// TIA Portal V17 export
// export: Created 2023-02-13T11:16:51.9785059Z, ExportSetting WithDefaults, DisplayName Totally Integrated Automation Portal, DisplayVersion V17, DisplayName TIA Portal Openness, DisplayVersion V17, DisplayName TIA Portal Teamcenter Gateway, DisplayVersion V17, DisplayName TIA Portal Version Control Interface, DisplayVersion V17, DisplayName SINAMICS Startdrive Advanced, DisplayVersion V17, DisplayName SINAMICS Startdrive G130, G150, S120, S150, SINAMICS MV, S210, DisplayVersion V17, DisplayName SINAMICS Startdrive G110M, G120, G120C, G120D, G120P, G115D, DisplayVersion V17, DisplayName STEP 7 Professional, DisplayVersion V17, DisplayName STEP 7 Safety, DisplayVersion V17, DisplayName WinCC Professional, DisplayVersion V17
FUNCTION_BLOCK "BFT_Type5"   // FB355, LAD
{ S7_Optimized_Access := 'TRUE' }
VERSION : 0.1
// Buffer Tank Vinegar
// stored: AutoNumber false, IsIECCheckEnabled false, IsRetainMemResEnabled false, MemoryReserve 100, SetENOAutomatically false, UDAEnableTagReadback false
   VAR_INPUT
      "IN_FBAV.01" : Bool := FALSE;   // Tank Flushing Water Valve
      "IN_FBAV.02" : Bool := FALSE;   // Tank CIP Top Inlet Valve
      "IN_FBAV.03" : Bool := FALSE;   // Tank Tank Outlet Valve
      "IN_FBSV.01" : Bool := FALSE;   // SV Diaphragm Pump Inlet Material
      IN_LT01 : Real;   // Tank Level Transmitter
      "IN_FBP.01" : Bool := FALSE;   // Transfer Pump
      "IN_P.01-Speed" : Real;   // Transfer Pump AV Speed
      DosePumpSpeed : Real;
      "DoseON-OFF" : Bool := FALSE;
      "DosePumpON-OFF" : Bool := FALSE;
      CIPPulse : Bool := FALSE;
      CIP_Supply_ON : Bool;
      CIP_Busy : Bool;   // Line CIP in USE
      LineTrf_OK : Bool := FALSE;
      LineFlush_OK : Bool;
      LCS_Start : Bool;   // Start Command from LCS
      LCS_Stop : Bool;   // Stop Command from LCS
   END_VAR
   VAR_OUTPUT
      "OUT_AV.01" : Bool := FALSE;   // Tank Flushing Water Valve
      "OUT_AV.02" : Bool := FALSE;   // Tank CIP Top Inlet Valve
      "OUT_AV.03" : Bool := FALSE;   // Tank Tank Outlet Valve
      "OUT_AV.06" : Bool := FALSE;   // Tank Tank Outlet Valve
      "OUT_P.01" : Bool := FALSE;   // Transfer Pump
      "OUT_P.01-Speed" : Real;   // Transfer Pump AV Speed
      "OUT_SV.01" : Bool := FALSE;   // SV Diaphragm Pump Inlet Material
      OUT_CIPTank_AVOpen : Bool;
   END_VAR
   VAR
      Cmd { ExternalVisible := 'False'} : Struct
         Inload { ExternalVisible := 'False'} : Bool;   // Start Loading
         RaadyForMix { ExternalVisible := 'False'} : Bool;   // Tank Ready for Blending
         Tank_CIP_Req { ExternalVisible := 'False'} : Bool;
         Flush_Select { ExternalVisible := 'False'} : Byte;
         Flushing { ExternalVisible := 'False'} : Bool;   // Water Flushing
      END_STRUCT;
      Param { ExternalVisible := 'False'} : Struct
         SP_Level_LL { ExternalVisible := 'False'} : Real := 10.0;
         SP_Level_ML { ExternalVisible := 'False'} : Real := 80.0;
         SP_Level_HL { ExternalVisible := 'False'} : Real := 100.0;
         L_Hi_Lim { ExternalVisible := 'False'} : Real := 100.0;
         L_Lo_Lim { ExternalVisible := 'False'} : Real := 0.0;
         L_Hys { ExternalVisible := 'False'} : Real := 5.0;
         FlushingTime { ExternalVisible := 'False'} : Time := T#10s;
         CIP_Trf_SP_Speed { ExternalVisible := 'False'} : Real := 80.0;
         CIP_Ret_ON_SP { ExternalVisible := 'False'} : Real := 5.0;
         CIP_Ret_OFF_SP { ExternalVisible := 'False'} : Real;
      END_STRUCT;
      State { ExternalVisible := 'False'} : Struct   // Tank in loading state
         Tank_inloading { ExternalVisible := 'False'} : Bool;
         Tank_inRawDose { ExternalVisible := 'False'} : Bool;
         Tank_inCIP { ExternalVisible := 'False'} : Bool;
         Line_inCIP { ExternalVisible := 'False'} : Bool;
         Flushing { ExternalVisible := 'False'} : Bool;
         Tank_LL { ExternalVisible := 'False'} : Bool;
         Tank_ML { ExternalVisible := 'False'} : Bool;
         Tank_HL { ExternalVisible := 'False'} : Bool;
         Inload_Enable { ExternalVisible := 'False'} : Bool;
         Tank_CIP_Enable { ExternalVisible := 'False'} : Bool;
         Line_CIP_Enable { ExternalVisible := 'False'} : Bool;
         Flushing_Enable { ExternalVisible := 'False'} : Bool;
         Flush_selected { ExternalVisible := 'False'} : Byte;
         CIP_Request_OK { ExternalVisible := 'False'} : Bool;
         CIP_ReturnON { ExternalVisible := 'False'} : Bool;
         Ready_For_Transfer { ExternalVisible := 'False'} : Bool;   // Tank Ready for Transfer to Blending
         Ready_For_Transfer_EN { ExternalVisible := 'False'} : Bool;   // Tank Ready for Transfer to Blending
         Transfer_to_Blend { ExternalVisible := 'False'} : Bool;
         Status { ExternalVisible := 'False'} : Int;
      END_STRUCT;
      alwaysON : Bool;
      L_Hys_Abs : Real;
      Hys_Level_HL : Real;
      Hys_Level_ML : Real;
      Hys_Level_LL : Real;
      r : Struct
         PosE1 : Bool;
         PosE2 : Bool;
         PosE3 : Bool;
         PosE4 : Bool;
         PosE5 : Bool;
         PosE6 : Bool;
         PosE7 : Bool;
         PosE8 : Bool;
         PosE9 : Bool;
         PosE10 : Bool;
         PosE11 : Bool;
         PosE12 : Bool;
         PosE13 : Bool;
         PosE14 : Bool;
         PosE15 : Bool;
         PosE16 : Bool;
         PosE17 : Bool;
         PosE18 : Bool;
         PosE19 : Bool;
         PosE20 : Bool;
         PosE21 : Bool;
         PosE22 : Bool;
         PosE23 : Bool;
         PosE24 : Bool;
         PosE25 : Bool;
         PosE26 : Bool;
         PosE27 : Bool;
         PosE28 : Bool;
         PosE29 : Bool;
         PosE30 : Bool;
         PosE31 : Bool;
         PosE32 : Bool;
      END_STRUCT;
      Actuator : Struct
         AV_Outlet : Bool;
         TransferPump : Bool;
         FlushPump : Bool;
         CV_Steam : Bool;
         Pump : Bool;
         Agitator_level : Bool;
         LCS_OnOff : Bool;
      END_STRUCT;
      FlushingTim : TON_TIME;
   END_VAR
   VAR_TEMP   // added for the SCL form of the ladder/FBD networks
      _w1 : Bool;
      _w2 : Bool;
      _w3 : Bool;
      _w4 : Bool;
      _w5 : Bool;
      _w6 : Bool;
   END_VAR
BEGIN

REGION Network 1: Always_ON
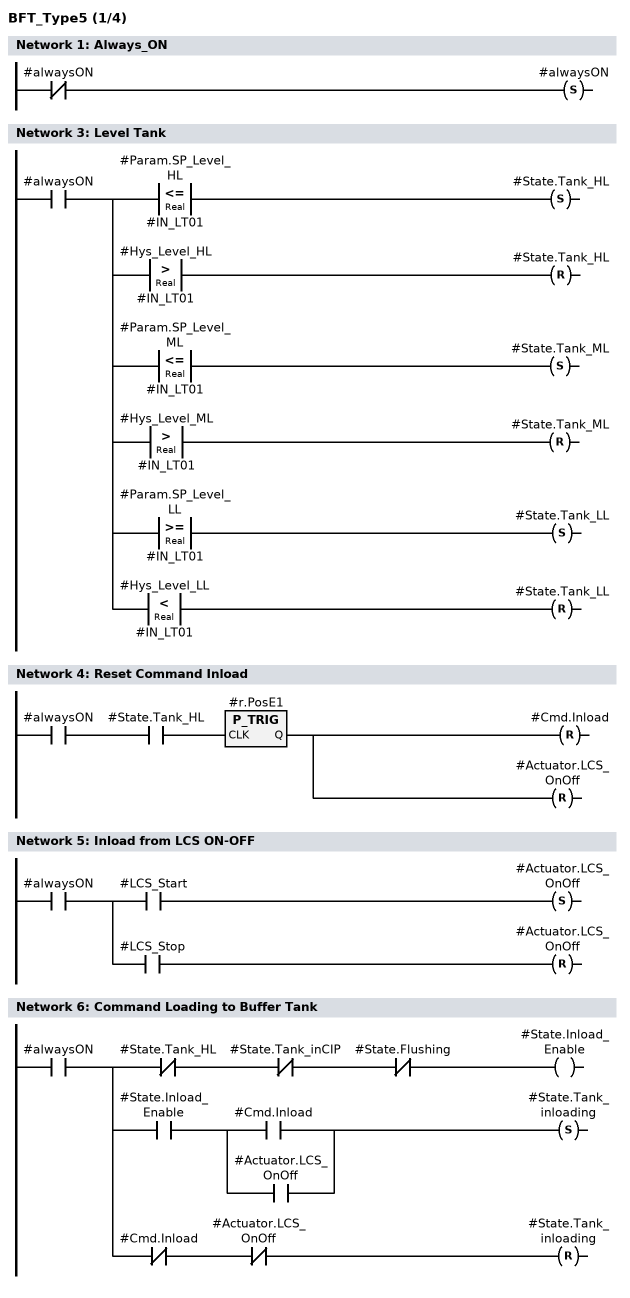
   RUNG wire#powerrail
      I_Contact( #alwaysON )
      S_Coil( #alwaysON )
   END_RUNG
   // the same network as SCL:
   IF NOT #alwaysON THEN #alwaysON := TRUE; END_IF;
END_REGION

NETWORK
TITLE = Hys Calculation
//Level Hys Absolute
      L     #Param.L_Hi_Lim;
      L     #Param.L_Lo_Lim;
      -R;
      L     100.0;
      /R;
      L     #Param.L_Hys;
      *R;
      T     #L_Hys_Abs;
//Tank High Level
      L     #Param.SP_Level_HL;
      L     #L_Hys_Abs;
      -R;
      T     #Hys_Level_HL;
//Tank Mid Level
      L     #Param.SP_Level_ML;
      L     #L_Hys_Abs;
      -R;
      T     #Hys_Level_ML;
//Tank Low Level
      L     #Param.SP_Level_LL;
      L     #L_Hys_Abs;
      +R;
      T     #Hys_Level_LL;


REGION Network 3: Level Tank
   RUNG wire#powerrail
      Contact( #alwaysON )
      wire#w1
      { S7_Templates := "SrcType := Real" } LE_Contact(in1 := #Param.SP_Level_HL, in2 := #IN_LT01)
      S_Coil( #State.Tank_HL )
   END_RUNG
   RUNG wire#w1
      { S7_Templates := "SrcType := Real" } GT_Contact(in1 := #Hys_Level_HL, in2 := #IN_LT01)
      R_Coil( #State.Tank_HL )
   END_RUNG
   RUNG wire#w1
      { S7_Templates := "SrcType := Real" } LE_Contact(in1 := #Param.SP_Level_ML, in2 := #IN_LT01)
      S_Coil( #State.Tank_ML )
   END_RUNG
   RUNG wire#w1
      { S7_Templates := "SrcType := Real" } GT_Contact(in1 := #Hys_Level_ML, in2 := #IN_LT01)
      R_Coil( #State.Tank_ML )
   END_RUNG
   RUNG wire#w1
      { S7_Templates := "SrcType := Real" } GE_Contact(in1 := #Param.SP_Level_LL, in2 := #IN_LT01)
      S_Coil( #State.Tank_LL )
   END_RUNG
   RUNG wire#w1
      { S7_Templates := "SrcType := Real" } LT_Contact(in1 := #Hys_Level_LL, in2 := #IN_LT01)
      R_Coil( #State.Tank_LL )
   END_RUNG
   // the same network as SCL:
   IF #alwaysON AND (#Param.SP_Level_HL <= #IN_LT01) THEN #State.Tank_HL := TRUE; END_IF;
   IF #alwaysON AND (#Hys_Level_HL > #IN_LT01) THEN #State.Tank_HL := FALSE; END_IF;
   IF #alwaysON AND (#Param.SP_Level_ML <= #IN_LT01) THEN #State.Tank_ML := TRUE; END_IF;
   IF #alwaysON AND (#Hys_Level_ML > #IN_LT01) THEN #State.Tank_ML := FALSE; END_IF;
   IF #alwaysON AND (#Param.SP_Level_LL >= #IN_LT01) THEN #State.Tank_LL := TRUE; END_IF;
   IF #alwaysON AND (#Hys_Level_LL < #IN_LT01) THEN #State.Tank_LL := FALSE; END_IF;
END_REGION

REGION Network 4: Reset Command Inload
   RUNG wire#powerrail
      Contact( #alwaysON )
      Contact( #State.Tank_HL )
      P_Trig( #r.PosE1 )
      wire#w1
      R_Coil( #Cmd.Inload )
   END_RUNG
   RUNG wire#w1
      R_Coil( #Actuator.LCS_OnOff )
   END_RUNG
   // the same network as SCL:
   #_w1 := #alwaysON AND #State.Tank_HL;
   #_w2 := #_w1 AND NOT #r.PosE1;   // rising edge
   #r.PosE1 := #_w1;
   IF #_w2 THEN
       #Cmd.Inload := FALSE;
       #Actuator.LCS_OnOff := FALSE;
   END_IF;
END_REGION

REGION Network 5: Inload from LCS ON-OFF
   RUNG wire#powerrail
      Contact( #alwaysON )
      wire#w1
      Contact( #LCS_Start )
      S_Coil( #Actuator.LCS_OnOff )
   END_RUNG
   RUNG wire#w1
      Contact( #LCS_Stop )
      R_Coil( #Actuator.LCS_OnOff )
   END_RUNG
   // the same network as SCL:
   IF #alwaysON AND #LCS_Start THEN #Actuator.LCS_OnOff := TRUE; END_IF;
   IF #alwaysON AND #LCS_Stop THEN #Actuator.LCS_OnOff := FALSE; END_IF;
END_REGION

REGION Network 6: Command Loading to Buffer Tank
   RUNG wire#powerrail
      Contact( #alwaysON )
      wire#w1
      I_Contact( #State.Tank_HL )
      I_Contact( #State.Tank_inCIP )
      I_Contact( #State.Flushing )
      Coil( #State.Inload_Enable )
   END_RUNG
   RUNG wire#w1
      Contact( #State.Inload_Enable )
      wire#w2
      Contact( #Cmd.Inload )
      wire#w3
      S_Coil( #State.Tank_inloading )
   END_RUNG
   RUNG wire#w2
      Contact( #Actuator.LCS_OnOff )
   END_RUNG wire#w3
   RUNG wire#w1
      I_Contact( #Cmd.Inload )
      I_Contact( #Actuator.LCS_OnOff )
      R_Coil( #State.Tank_inloading )
   END_RUNG
   // the same network as SCL:
   #State.Inload_Enable := #alwaysON AND NOT #State.Tank_HL AND NOT #State.Tank_inCIP AND NOT #State.Flushing;
   IF #alwaysON AND #State.Inload_Enable AND (#Cmd.Inload OR #Actuator.LCS_OnOff) THEN
       #State.Tank_inloading := TRUE;
   END_IF;
   IF #alwaysON AND NOT #Cmd.Inload AND NOT #Actuator.LCS_OnOff THEN #State.Tank_inloading := FALSE; END_IF;
END_REGION

REGION Network 7: Choose Flush Destination
   // #Cmd.Flush_Select.%X0 = T-20.00
   // #Cmd.Flush_Select.%X1 = T-21.00
   // #Cmd.Flush_Select.%X2 = T-30.00
   // #Cmd.Flush_Select.%X3 = T-31.00
   // #Cmd.Flush_Select.%X4 = Drain
   // #Cmd.Flush_Select.%X5 = Flush_Selected
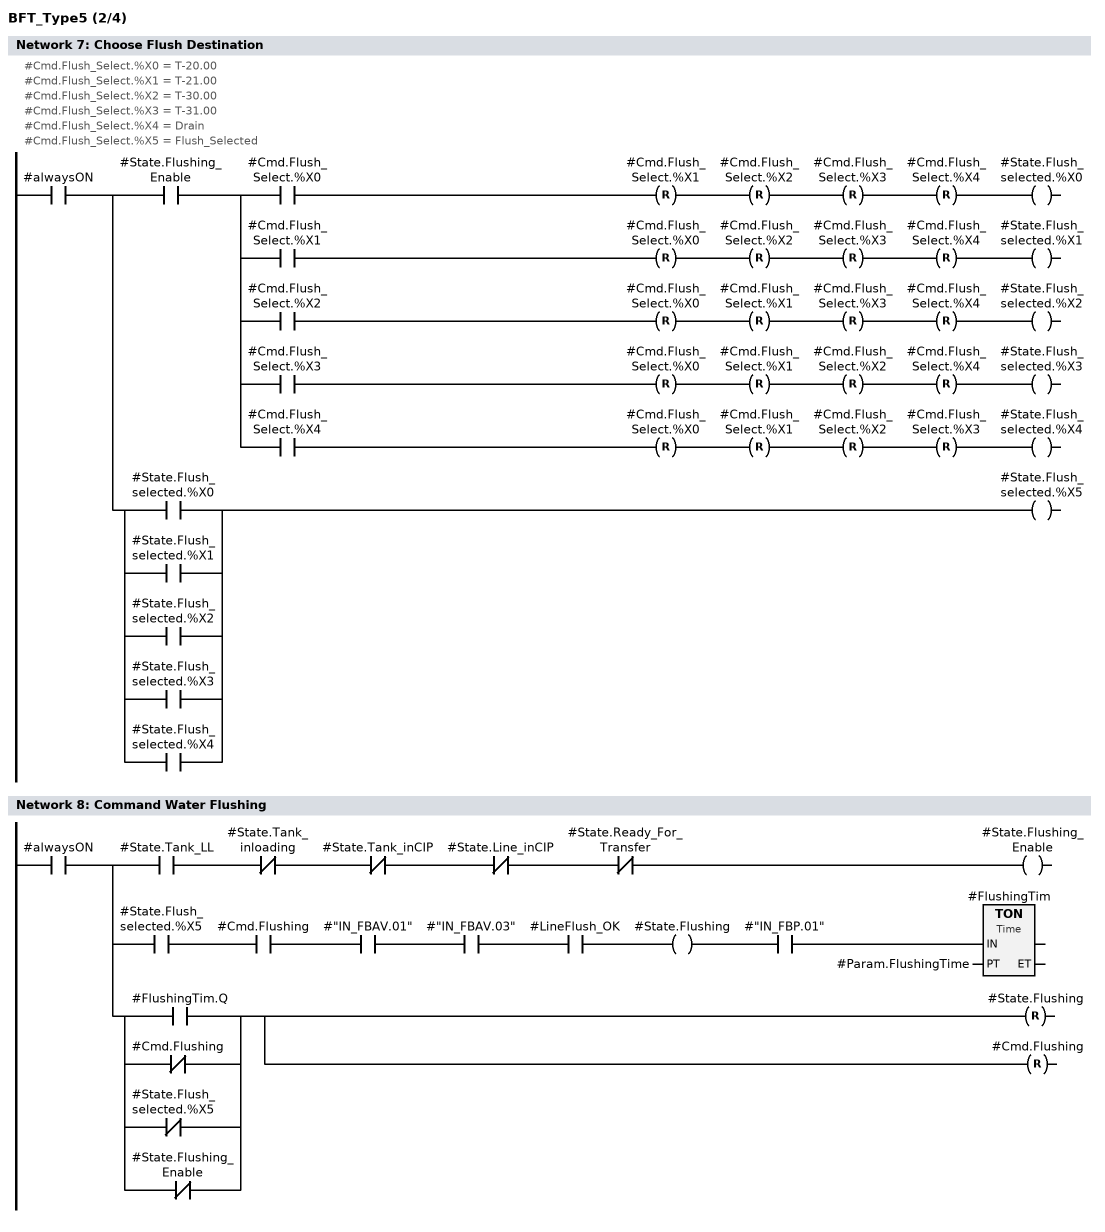
   RUNG wire#powerrail
      Contact( #alwaysON )
      wire#w1
      Contact( #State.Flushing_Enable )
      wire#w2
      Contact( #Cmd.Flush_Select.%X0 )
      R_Coil( #Cmd.Flush_Select.%X1 )
      R_Coil( #Cmd.Flush_Select.%X2 )
      R_Coil( #Cmd.Flush_Select.%X3 )
      R_Coil( #Cmd.Flush_Select.%X4 )
      Coil( #State.Flush_selected.%X0 )
   END_RUNG
   RUNG wire#w2
      Contact( #Cmd.Flush_Select.%X1 )
      R_Coil( #Cmd.Flush_Select.%X0 )
      R_Coil( #Cmd.Flush_Select.%X2 )
      R_Coil( #Cmd.Flush_Select.%X3 )
      R_Coil( #Cmd.Flush_Select.%X4 )
      Coil( #State.Flush_selected.%X1 )
   END_RUNG
   RUNG wire#w2
      Contact( #Cmd.Flush_Select.%X2 )
      R_Coil( #Cmd.Flush_Select.%X0 )
      R_Coil( #Cmd.Flush_Select.%X1 )
      R_Coil( #Cmd.Flush_Select.%X3 )
      R_Coil( #Cmd.Flush_Select.%X4 )
      Coil( #State.Flush_selected.%X2 )
   END_RUNG
   RUNG wire#w2
      Contact( #Cmd.Flush_Select.%X3 )
      R_Coil( #Cmd.Flush_Select.%X0 )
      R_Coil( #Cmd.Flush_Select.%X1 )
      R_Coil( #Cmd.Flush_Select.%X2 )
      R_Coil( #Cmd.Flush_Select.%X4 )
      Coil( #State.Flush_selected.%X3 )
   END_RUNG
   RUNG wire#w2
      Contact( #Cmd.Flush_Select.%X4 )
      R_Coil( #Cmd.Flush_Select.%X0 )
      R_Coil( #Cmd.Flush_Select.%X1 )
      R_Coil( #Cmd.Flush_Select.%X2 )
      R_Coil( #Cmd.Flush_Select.%X3 )
      Coil( #State.Flush_selected.%X4 )
   END_RUNG
   RUNG wire#w1
      Contact( #State.Flush_selected.%X0 )
      wire#w3
      Coil( #State.Flush_selected.%X5 )
   END_RUNG
   RUNG wire#w1
      Contact( #State.Flush_selected.%X1 )
   END_RUNG wire#w3
   RUNG wire#w1
      Contact( #State.Flush_selected.%X2 )
   END_RUNG wire#w3
   RUNG wire#w1
      Contact( #State.Flush_selected.%X3 )
   END_RUNG wire#w3
   RUNG wire#w1
      Contact( #State.Flush_selected.%X4 )
   END_RUNG wire#w3
   // the same network as SCL:
   #_w1 := #alwaysON AND #State.Flushing_Enable;
   #_w2 := #_w1 AND #Cmd.Flush_Select.%X0;
   IF #_w2 THEN
       #Cmd.Flush_Select.%X1 := FALSE;
       #Cmd.Flush_Select.%X2 := FALSE;
       #Cmd.Flush_Select.%X3 := FALSE;
       #Cmd.Flush_Select.%X4 := FALSE;
   END_IF;
   #State.Flush_selected.%X0 := #_w2;
   #_w3 := #_w1 AND #Cmd.Flush_Select.%X1;
   IF #_w3 THEN
       #Cmd.Flush_Select.%X0 := FALSE;
       #Cmd.Flush_Select.%X2 := FALSE;
       #Cmd.Flush_Select.%X3 := FALSE;
       #Cmd.Flush_Select.%X4 := FALSE;
   END_IF;
   #State.Flush_selected.%X1 := #_w3;
   #_w4 := #_w1 AND #Cmd.Flush_Select.%X2;
   IF #_w4 THEN
       #Cmd.Flush_Select.%X0 := FALSE;
       #Cmd.Flush_Select.%X1 := FALSE;
       #Cmd.Flush_Select.%X3 := FALSE;
       #Cmd.Flush_Select.%X4 := FALSE;
   END_IF;
   #State.Flush_selected.%X2 := #_w4;
   #_w5 := #_w1 AND #Cmd.Flush_Select.%X3;
   IF #_w5 THEN
       #Cmd.Flush_Select.%X0 := FALSE;
       #Cmd.Flush_Select.%X1 := FALSE;
       #Cmd.Flush_Select.%X2 := FALSE;
       #Cmd.Flush_Select.%X4 := FALSE;
   END_IF;
   #State.Flush_selected.%X3 := #_w5;
   #_w6 := #_w1 AND #Cmd.Flush_Select.%X4;
   IF #_w6 THEN
       #Cmd.Flush_Select.%X0 := FALSE;
       #Cmd.Flush_Select.%X1 := FALSE;
       #Cmd.Flush_Select.%X2 := FALSE;
       #Cmd.Flush_Select.%X3 := FALSE;
   END_IF;
   #State.Flush_selected.%X4 := #_w6;
   #State.Flush_selected.%X5 := #alwaysON AND (#State.Flush_selected.%X0 OR #State.Flush_selected.%X1 OR #State.Flush_selected.%X2 OR #State.Flush_selected.%X3 OR #State.Flush_selected.%X4);
END_REGION

REGION Network 8: Command Water Flushing
   RUNG wire#powerrail
      Contact( #alwaysON )
      wire#w1
      Contact( #State.Tank_LL )
      I_Contact( #State.Tank_inloading )
      I_Contact( #State.Tank_inCIP )
      I_Contact( #State.Line_inCIP )
      I_Contact( #State.Ready_For_Transfer )
      Coil( #State.Flushing_Enable )
   END_RUNG
   RUNG wire#w1
      Contact( #State.Flush_selected.%X5 )
      Contact( #Cmd.Flushing )
      Contact( #"IN_FBAV.01" )
      Contact( #"IN_FBAV.03" )
      Contact( #LineFlush_OK )
      Coil( #State.Flushing )
      Contact( #"IN_FBP.01" )
      { S7_Templates := "time_type := Time" } #FlushingTim.TON(pt := #Param.FlushingTime, et =>)
   END_RUNG
   RUNG wire#w1
      Contact( #FlushingTim.Q )
      wire#w2
      R_Coil( #State.Flushing )
   END_RUNG
   RUNG wire#w1
      I_Contact( #Cmd.Flushing )
   END_RUNG wire#w2
   RUNG wire#w1
      I_Contact( #State.Flush_selected.%X5 )
   END_RUNG wire#w2
   RUNG wire#w1
      I_Contact( #State.Flushing_Enable )
   END_RUNG wire#w2
   RUNG wire#w2
      R_Coil( #Cmd.Flushing )
   END_RUNG
   // the same network as SCL:
   #State.Flushing_Enable := #alwaysON AND #State.Tank_LL AND NOT #State.Tank_inloading AND NOT #State.Tank_inCIP AND NOT #State.Line_inCIP AND NOT #State.Ready_For_Transfer;
   #State.Flushing := #alwaysON AND #State.Flush_selected.%X5 AND #Cmd.Flushing AND #"IN_FBAV.01" AND #"IN_FBAV.03" AND #LineFlush_OK;
   #FlushingTim(IN := #State.Flushing AND #"IN_FBP.01", PT := #Param.FlushingTime);   // TON
   IF #alwaysON AND (#FlushingTim.Q OR NOT #Cmd.Flushing OR NOT #State.Flush_selected.%X5 OR NOT #State.Flushing_Enable) THEN
       #State.Flushing := FALSE;
       #Cmd.Flushing := FALSE;
   END_IF;
END_REGION

REGION Network 9: Flushing Destination AV and Pump
   // #Cmd.Flush_Select.%X0 = T-20.00
   // #Cmd.Flush_Select.%X1 = T-21.00
   // #Cmd.Flush_Select.%X2 = T-30.00
   // #Cmd.Flush_Select.%X3 = T-31.00
   // #Cmd.Flush_Select.%X4 = Drain
   // #Cmd.Flush_Select.%X5 = Flush_Selected
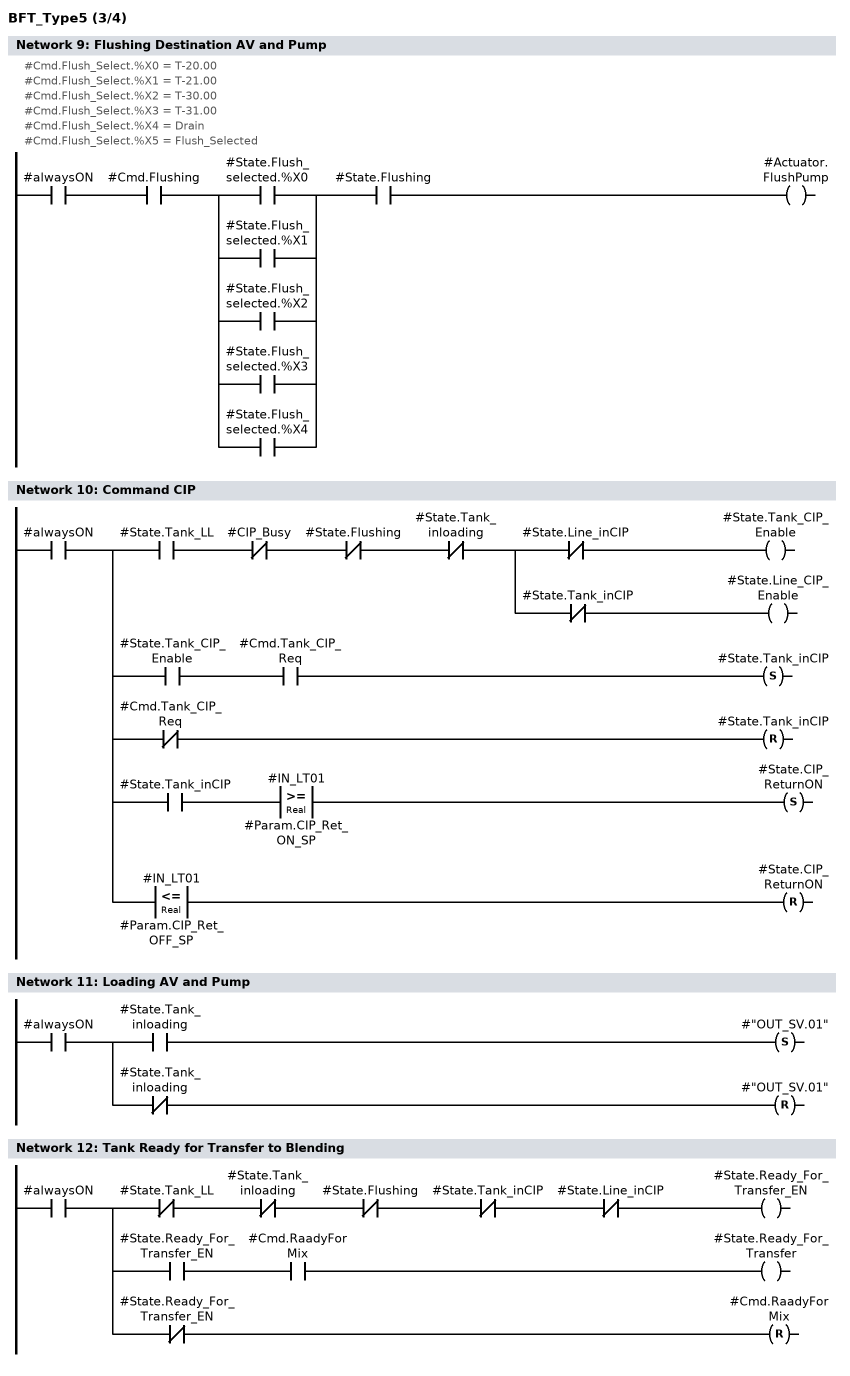
   RUNG wire#powerrail
      Contact( #alwaysON )
      Contact( #Cmd.Flushing )
      wire#w1
      Contact( #State.Flush_selected.%X0 )
      wire#w2
      Contact( #State.Flushing )
      Coil( #Actuator.FlushPump )
   END_RUNG
   RUNG wire#w1
      Contact( #State.Flush_selected.%X1 )
   END_RUNG wire#w2
   RUNG wire#w1
      Contact( #State.Flush_selected.%X2 )
   END_RUNG wire#w2
   RUNG wire#w1
      Contact( #State.Flush_selected.%X3 )
   END_RUNG wire#w2
   RUNG wire#w1
      Contact( #State.Flush_selected.%X4 )
   END_RUNG wire#w2
   // the same network as SCL:
   #Actuator.FlushPump := #alwaysON AND #Cmd.Flushing AND (#State.Flush_selected.%X0 OR #State.Flush_selected.%X1 OR #State.Flush_selected.%X2 OR #State.Flush_selected.%X3 OR #State.Flush_selected.%X4) AND #State.Flushing;
END_REGION

REGION Network 10: Command CIP
   RUNG wire#powerrail
      Contact( #alwaysON )
      wire#w1
      Contact( #State.Tank_LL )
      I_Contact( #CIP_Busy )
      I_Contact( #State.Flushing )
      I_Contact( #State.Tank_inloading )
      wire#w2
      I_Contact( #State.Line_inCIP )
      Coil( #State.Tank_CIP_Enable )
   END_RUNG
   RUNG wire#w2
      I_Contact( #State.Tank_inCIP )
      Coil( #State.Line_CIP_Enable )
   END_RUNG
   RUNG wire#w1
      Contact( #State.Tank_CIP_Enable )
      Contact( #Cmd.Tank_CIP_Req )
      S_Coil( #State.Tank_inCIP )
   END_RUNG
   RUNG wire#w1
      I_Contact( #Cmd.Tank_CIP_Req )
      R_Coil( #State.Tank_inCIP )
   END_RUNG
   RUNG wire#w1
      Contact( #State.Tank_inCIP )
      { S7_Templates := "SrcType := Real" } GE_Contact(in1 := #IN_LT01, in2 := #Param.CIP_Ret_ON_SP)
      S_Coil( #State.CIP_ReturnON )
   END_RUNG
   RUNG wire#w1
      { S7_Templates := "SrcType := Real" } LE_Contact(in1 := #IN_LT01, in2 := #Param.CIP_Ret_OFF_SP)
      R_Coil( #State.CIP_ReturnON )
   END_RUNG
   // the same network as SCL:
   #_w1 := #alwaysON AND #State.Tank_LL AND NOT #CIP_Busy AND NOT #State.Flushing AND NOT #State.Tank_inloading;
   #State.Tank_CIP_Enable := #_w1 AND NOT #State.Line_inCIP;
   #State.Line_CIP_Enable := #_w1 AND NOT #State.Tank_inCIP;
   IF #alwaysON AND #State.Tank_CIP_Enable AND #Cmd.Tank_CIP_Req THEN #State.Tank_inCIP := TRUE; END_IF;
   IF #alwaysON AND NOT #Cmd.Tank_CIP_Req THEN #State.Tank_inCIP := FALSE; END_IF;
   IF #alwaysON AND #State.Tank_inCIP AND (#IN_LT01 >= #Param.CIP_Ret_ON_SP) THEN
       #State.CIP_ReturnON := TRUE;
   END_IF;
   IF #alwaysON AND (#IN_LT01 <= #Param.CIP_Ret_OFF_SP) THEN #State.CIP_ReturnON := FALSE; END_IF;
END_REGION

REGION Network 11: Loading AV and Pump
   RUNG wire#powerrail
      Contact( #alwaysON )
      wire#w1
      Contact( #State.Tank_inloading )
      S_Coil( #"OUT_SV.01" )
   END_RUNG
   RUNG wire#w1
      I_Contact( #State.Tank_inloading )
      R_Coil( #"OUT_SV.01" )
   END_RUNG
   // the same network as SCL:
   IF #alwaysON AND #State.Tank_inloading THEN #"OUT_SV.01" := TRUE; END_IF;
   IF #alwaysON AND NOT #State.Tank_inloading THEN #"OUT_SV.01" := FALSE; END_IF;
END_REGION

REGION Network 12: Tank Ready for Transfer to Blending
   RUNG wire#powerrail
      Contact( #alwaysON )
      wire#w1
      I_Contact( #State.Tank_LL )
      I_Contact( #State.Tank_inloading )
      I_Contact( #State.Flushing )
      I_Contact( #State.Tank_inCIP )
      I_Contact( #State.Line_inCIP )
      Coil( #State.Ready_For_Transfer_EN )
   END_RUNG
   RUNG wire#w1
      Contact( #State.Ready_For_Transfer_EN )
      Contact( #Cmd.RaadyForMix )
      Coil( #State.Ready_For_Transfer )
   END_RUNG
   RUNG wire#w1
      I_Contact( #State.Ready_For_Transfer_EN )
      R_Coil( #Cmd.RaadyForMix )
   END_RUNG
   // the same network as SCL:
   #State.Ready_For_Transfer_EN := #alwaysON AND NOT #State.Tank_LL AND NOT #State.Tank_inloading AND NOT #State.Flushing AND NOT #State.Tank_inCIP AND NOT #State.Line_inCIP;
   #State.Ready_For_Transfer := #alwaysON AND #State.Ready_For_Transfer_EN AND #Cmd.RaadyForMix;
   IF #alwaysON AND NOT #State.Ready_For_Transfer_EN THEN #Cmd.RaadyForMix := FALSE; END_IF;
END_REGION

REGION Network 13: Transfer to Blending AV and Pump
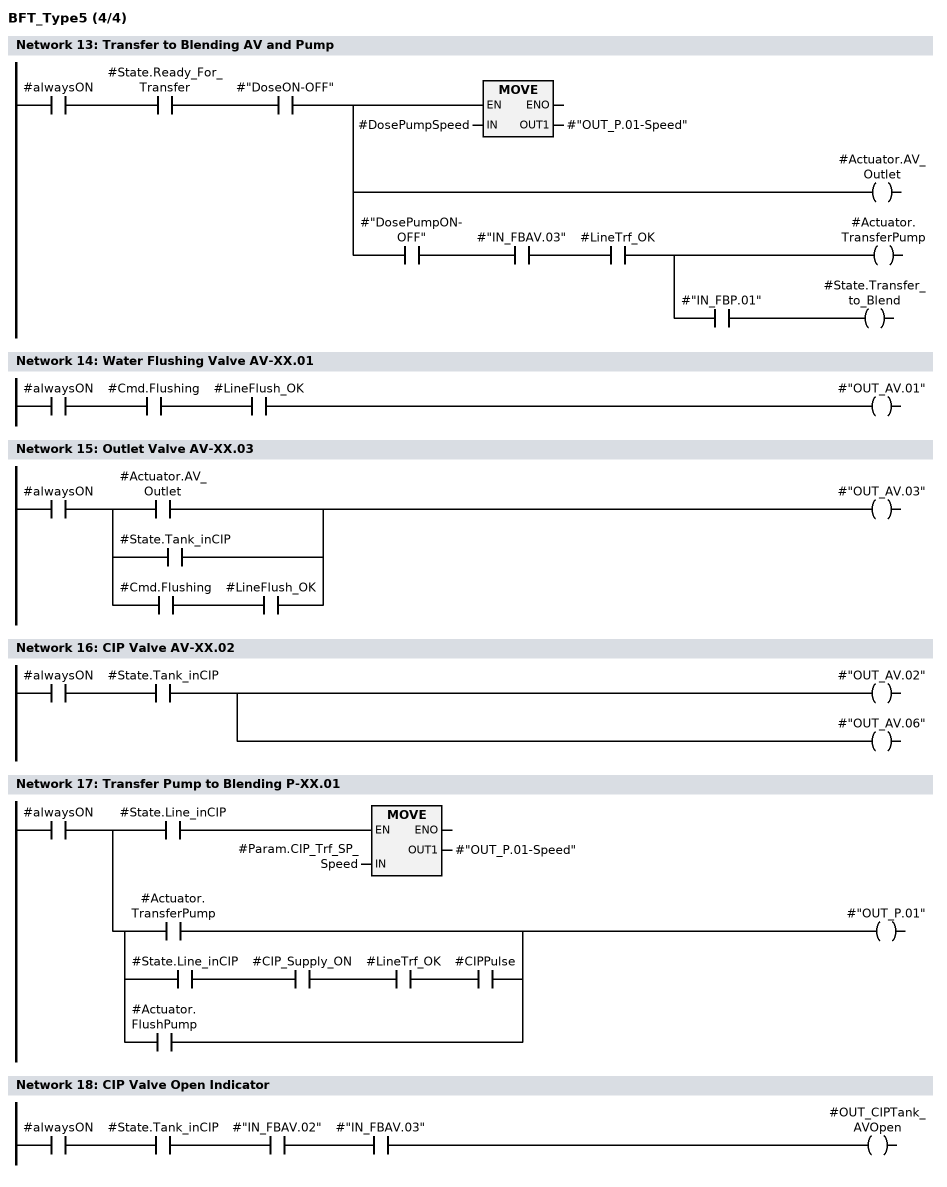
   RUNG wire#powerrail
      Contact( #alwaysON )
      Contact( #State.Ready_For_Transfer )
      Contact( #"DoseON-OFF" )
      wire#w1
      Move(in := #DosePumpSpeed, out1 => #"OUT_P.01-Speed")
   END_RUNG
   RUNG wire#w1
      Coil( #Actuator.AV_Outlet )
   END_RUNG
   RUNG wire#w1
      Contact( #"DosePumpON-OFF" )
      Contact( #"IN_FBAV.03" )
      Contact( #LineTrf_OK )
      wire#w2
      Coil( #Actuator.TransferPump )
   END_RUNG
   RUNG wire#w2
      Contact( #"IN_FBP.01" )
      Coil( #State.Transfer_to_Blend )
   END_RUNG
   // the same network as SCL:
   #_w1 := #alwaysON AND #State.Ready_For_Transfer AND #"DoseON-OFF";
   IF #_w1 THEN #"OUT_P.01-Speed" := #DosePumpSpeed; END_IF;
   #Actuator.AV_Outlet := #_w1;
   #Actuator.TransferPump := #_w1 AND #"DosePumpON-OFF" AND #"IN_FBAV.03" AND #LineTrf_OK;
   #State.Transfer_to_Blend := #Actuator.TransferPump AND #"IN_FBP.01";
END_REGION

REGION Network 14: Water Flushing Valve AV-XX.01
   RUNG wire#powerrail
      Contact( #alwaysON )
      Contact( #Cmd.Flushing )
      Contact( #LineFlush_OK )
      Coil( #"OUT_AV.01" )
   END_RUNG
   // the same network as SCL:
   #"OUT_AV.01" := #alwaysON AND #Cmd.Flushing AND #LineFlush_OK;
END_REGION

REGION Network 15: Outlet Valve AV-XX.03
   RUNG wire#powerrail
      Contact( #alwaysON )
      wire#w1
      Contact( #Actuator.AV_Outlet )
      wire#w2
      Coil( #"OUT_AV.03" )
   END_RUNG
   RUNG wire#w1
      Contact( #State.Tank_inCIP )
   END_RUNG wire#w2
   RUNG wire#w1
      Contact( #Cmd.Flushing )
      Contact( #LineFlush_OK )
   END_RUNG wire#w2
   // the same network as SCL:
   #"OUT_AV.03" := #alwaysON AND (#Actuator.AV_Outlet OR #State.Tank_inCIP OR (#Cmd.Flushing AND #LineFlush_OK));
END_REGION

REGION Network 16: CIP Valve AV-XX.02
   RUNG wire#powerrail
      Contact( #alwaysON )
      Contact( #State.Tank_inCIP )
      wire#w1
      Coil( #"OUT_AV.02" )
   END_RUNG
   RUNG wire#w1
      Coil( #"OUT_AV.06" )
   END_RUNG
   // the same network as SCL:
   #"OUT_AV.02" := #alwaysON AND #State.Tank_inCIP;
   #"OUT_AV.06" := #"OUT_AV.02";
END_REGION

REGION Network 17: Transfer Pump to Blending P-XX.01
   RUNG wire#powerrail
      Contact( #alwaysON )
      wire#w1
      Contact( #State.Line_inCIP )
      Move(in := #Param.CIP_Trf_SP_Speed, out1 => #"OUT_P.01-Speed")
   END_RUNG
   RUNG wire#w1
      Contact( #Actuator.TransferPump )
      wire#w2
      Coil( #"OUT_P.01" )
   END_RUNG
   RUNG wire#w1
      Contact( #State.Line_inCIP )
      Contact( #CIP_Supply_ON )
      Contact( #LineTrf_OK )
      Contact( #CIPPulse )
   END_RUNG wire#w2
   RUNG wire#w1
      Contact( #Actuator.FlushPump )
   END_RUNG wire#w2
   // the same network as SCL:
   IF #alwaysON AND #State.Line_inCIP THEN #"OUT_P.01-Speed" := #Param.CIP_Trf_SP_Speed; END_IF;
   #"OUT_P.01" := #alwaysON AND (#Actuator.TransferPump OR (#State.Line_inCIP AND #CIP_Supply_ON AND #LineTrf_OK AND #CIPPulse) OR #Actuator.FlushPump);
END_REGION

REGION Network 18: CIP Valve Open Indicator
   RUNG wire#powerrail
      Contact( #alwaysON )
      Contact( #State.Tank_inCIP )
      Contact( #"IN_FBAV.02" )
      Contact( #"IN_FBAV.03" )
      Coil( #OUT_CIPTank_AVOpen )
   END_RUNG
   // the same network as SCL:
   #OUT_CIPTank_AVOpen := #alwaysON AND #State.Tank_inCIP AND #"IN_FBAV.02" AND #"IN_FBAV.03";
END_REGION
END_FUNCTION_BLOCK
